RoboDK station: Assistive_UR5e.rdk

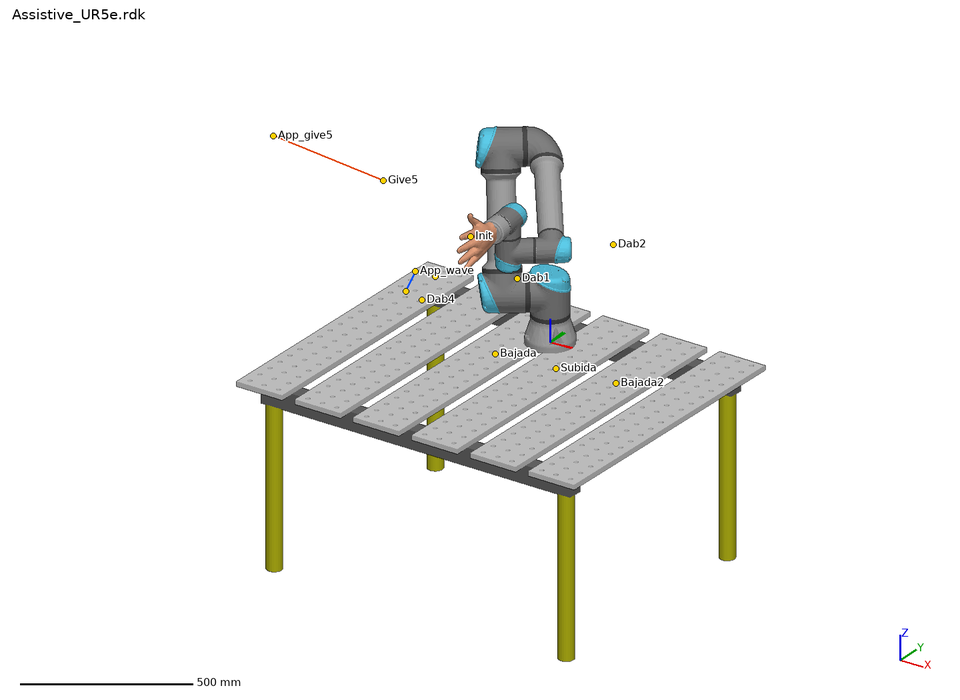
[picture v0: the station drawn from its stored meshes, robots at their saved joint values, targets as dots, program paths as lines]
Station Assistive_UR5e_SW (saved by RoboDK 5.9.2). Poses are relative to the parent item; angles as X-Y-Z fixed-axis rotations.
  - frame UR5e Base at (0, 0, 0) mm, rotated rx 0 ry 0 rz 5.71 deg
    - robot UR5e: 6 axes, payload 5 kg, reach 850 mm, repeatability 0.03 mm, weight 18.4 kg
        modified DH rows (alpha deg, a mm, theta deg, d mm): 0, 0, 0, 162.5; 90, 0, 180, 0; 0, 425, 0, 0; 0, 392.25, 0, 133.3; -90, 0, 0, 99.7; 90, 0, 180, 99.6
        joint limits [-360, -360, -360, -360, -360, -360] to [360, 360, 360, 360, 360, 360]; home [0, -90, -90, 0, 90, 0]; saved at [-57.836, -69.983, -134.335, -335.683, -302.164, 180]
      - tool Hand, TCP at (0, 0, 50) mm, size 54.8 x 155.9 x 193.5 mm, geometry from Hand.stl
  - frame World at (0, 0, 0) mm
    - object Table at (0, 0, 0) mm, size 1193.8 x 965.2 x 609.6 mm, geometry from welding_table.sld
    - target Init (Cartesian target) at (0, -400, 500) mm, rotated rx 90 ry 0 rz 0 deg; joints [-57.836, -85.391, -107.167, 172.559, -57.836, 0] of UR5e
    - target App_wave (Cartesian target) at (0, -680, 500) mm, rotated rx 90 ry 0 rz 0 deg; joints [75.444, 18.986, -92.472, -106.514, -75.444, 180] of UR5e
    - target Wave (Cartesian target) at (67.6, -676.63, 500) mm, rotated rx -120.53 ry -80.83 rz -46.18 deg; joints [-91.174, -132.208, -29.443, -171.146, -190.197, 124.748] of UR5e
    - target Bajada (Cartesian target) at (266.61, -656.75, 300) mm, rotated rx 168.48 ry -36.56 rz 9.52 deg; joints [-68.848, -118.561, -85.504, -41.08, -240.155, 207.874] of UR5e
    - target Subida (Cartesian target) at (465.62, -636.87, 300) mm, rotated rx 15.33 ry -52.65 rz 170.3 deg; joints [-57.574, -135.775, -73.382, 265.429, -135.289, -234.622] of UR5e
    - target Bajada2 (Cartesian target) at (664.63, -616.98, 300) mm, rotated rx 158.97 ry -63.45 rz 21.58 deg; joints [-45.449, -150.106, -44.369, -15.769, 124.078, -118.259] of UR5e
    - target Dab1 (Cartesian target) at (234.23, -501.09, 469.88) mm, rotated rx -88.57 ry 1.43 rz 89.43 deg; joints [-46.177, -123.095, -49.986, -188.777, 50.151, -177.384] of UR5e
    - target Dab2 (Cartesian target) at (487.14, -378.39, 601.54) mm, rotated rx 3.19 ry 2.8 rz 83.99 deg; joints [-31.988, -136.154, -45.027, 89.151, 93.729, 200.128] of UR5e
    - target Dab3 (Cartesian target) at (487.14, -378.39, 601.54) mm, rotated rx 92.17 ry 2.8 rz 83.99 deg; joints [-37.072, -101.911, -88.483, 8.002, 115.231, 176.178] of UR5e
    - target Dab4 (Cartesian target) at (-119.89, -474.77, 291.3) mm, rotated rx -18.93 ry -66.24 rz 24.97 deg; joints [-76.804, -121.175, -96.572, -201.012, 26.471, -205.994] of UR5e
    - target Shake (joint target) at (-300, -300, 200) mm, rotated rx 90 ry 0 rz 0 deg; joints [-129.97, -95.332, -131.473, -133.195, -129.97, 0] of UR5e
    - target Give5 (joint target) at (-380.86, -300, 533.82) mm, rotated rx 0 ry 0 rz 90 deg; joints [-125.814, -94.091, -116.939, 301.03, -90, 125.814] of UR5e
    - target App_give5 (joint target) at (-810.86, -238.62, 533.82) mm, rotated rx 0 ry 0 rz 90 deg; joints [-154.528, -143.977, -40.15, 274.127, -90, 154.528] of UR5e
    - target Wave2 (Cartesian target) at (0, -680, 500) mm, rotated rx 165.29 ry 0 rz 86.57 deg; joints [-81.878, -163.91, 50.211, -153.291, 104.409, 101.932] of UR5e
  - program Init (3 instructions, listed below)
  - program Hand_shake (5 instructions, listed below)
  - program Give_me_5! (5 instructions, listed below)
  - program MainProgram (4 instructions, listed below)
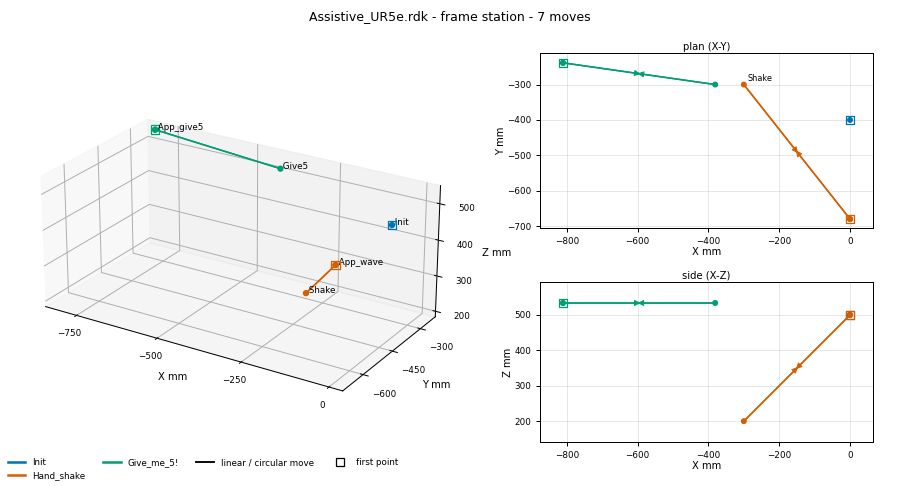
[picture p0: tool path of Assistive_UR5e.rdk in frame station, 7 of 7 moves have a stored position in this frame; points joined in program order, loops and branches not executed]

--- program Init (robot UR5e) ---
  Est. Ref.: UR5e Base
  Est. herr: Hand
  MoveJ (Init)

--- program Hand_shake (robot UR5e) ---
  Est. Ref.: UR5e Base
  Est. herr: Hand
  MoveL (App_shake) -> target App_wave
  MoveL (Shake)
  MoveL (App_shake) -> target App_wave

--- program Give_me_5! (robot UR5e) ---
  Est. Ref.: UR5e Base
  Est. herr: Hand
  MoveL (App_give5)
  MoveL (Give5)
  MoveL (App_give5)

--- program MainProgram (robot UR5e) ---
  Llamar Init
  Llamar Hand_shake
  Llamar Give_me_5!
  Llamar Init
